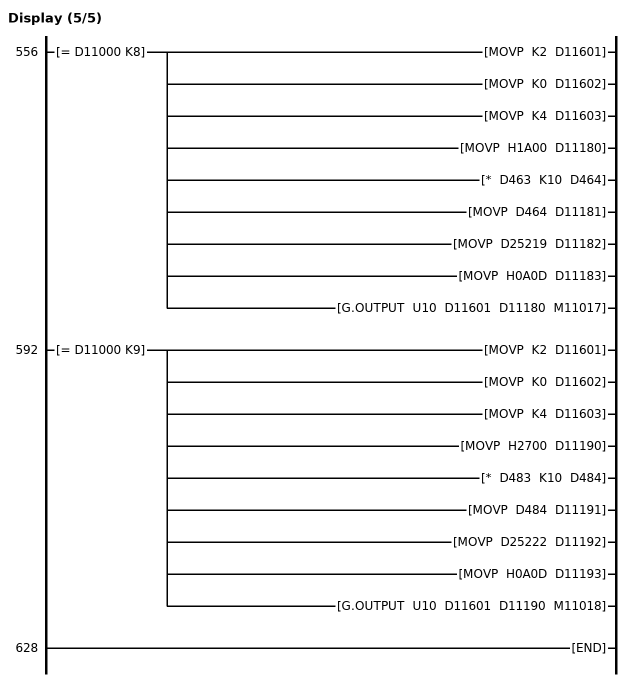
[picture p216: ladder of Display, rungs at steps 556 to 628]
556   LD=     D11000 K8
      MOVP    K2 D11601
      MOVP    K0 D11602
      MOVP    K4 D11603
      MOVP    H1A00 D11180
      *       D463 K10 D464
      MOVP    D464 D11181
      MOVP    D25219 D11182
      MOVP    H0A0D D11183
      G.OUTPUT U10 D11601 D11180 M11017
592   LD=     D11000 K9
      MOVP    K2 D11601
      MOVP    K0 D11602
      MOVP    K4 D11603
      MOVP    H2700 D11190
      *       D483 K10 D484
      MOVP    D484 D11191
      MOVP    D25222 D11192
      MOVP    H0A0D D11193
      G.OUTPUT U10 D11601 D11190 M11018
628   END
END_PROGRAM

PROGRAM door
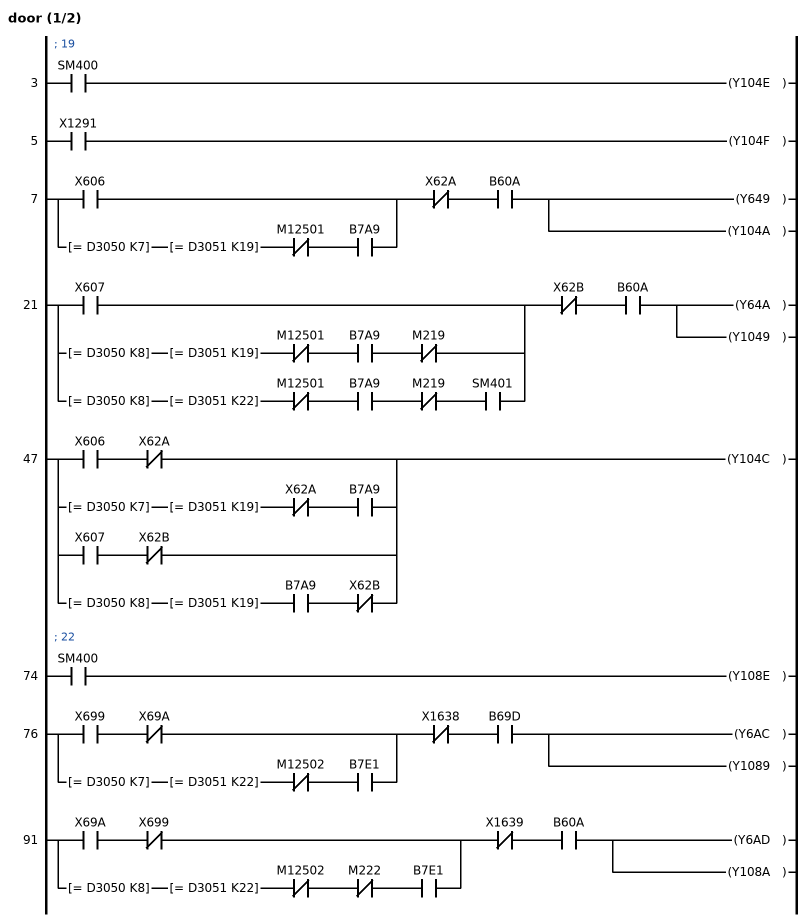
; 19
3     LD      SM400
      OUT     Y104E
5     LD      X1291
      OUT     Y104F
7     LD      X606
      LD=     D3050 K7
      AND=    D3051 K19
      ANI     M12501
      AND     B7A9
      ORB
      ANI     X62A
      AND     B60A
      OUT     Y649
      OUT     Y104A
21    LD      X607
      LD=     D3050 K8
      AND=    D3051 K19
      ANI     M12501
      AND     B7A9
      ANI     M219
      ORB
      LD=     D3050 K8
      AND=    D3051 K22
      ANI     M12501
      AND     B7A9
      ANI     M219
      AND     SM401
      ORB
      ANI     X62B
      AND     B60A
      OUT     Y64A
      OUT     Y1049
47    LD      X606
      ANI     X62A
      LD=     D3050 K7
      AND=    D3051 K19
      ANI     X62A
      AND     B7A9
      ORB
      LD      X607
      ANI     X62B
      ORB
      LD=     D3050 K8
      AND=    D3051 K19
      AND     B7A9
      ANI     X62B
      ORB
      OUT     Y104C
; 22
74    LD      SM400
      OUT     Y108E
76    LD      X699
      ANI     X69A
      LD=     D3050 K7
      AND=    D3051 K22
      ANI     M12502
      AND     B7E1
      ORB
      ANI     X1638
      AND     B69D
      OUT     Y6AC
      OUT     Y1089
91    LD      X69A
      ANI     X699
      LD=     D3050 K8
      AND=    D3051 K22
      ANI     M12502
      ANI     M222
      AND     B7E1
      ORB
      ANI     X1639
      AND     B60A
      OUT     Y6AD
      OUT     Y108A
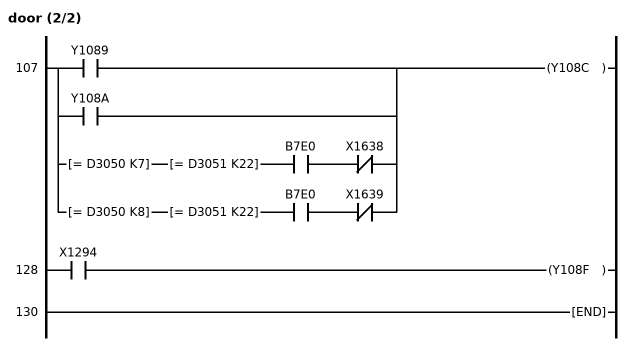
107   LD      Y1089
      OR      Y108A
      LD=     D3050 K7
      AND=    D3051 K22
      AND     B7E0
      ANI     X1638
      ORB
      LD=     D3050 K8
      AND=    D3051 K22
      AND     B7E0
      ANI     X1639
      ORB
      OUT     Y108C
128   LD      X1294
      OUT     Y108F
130   END
END_PROGRAM

PROGRAM enter_line
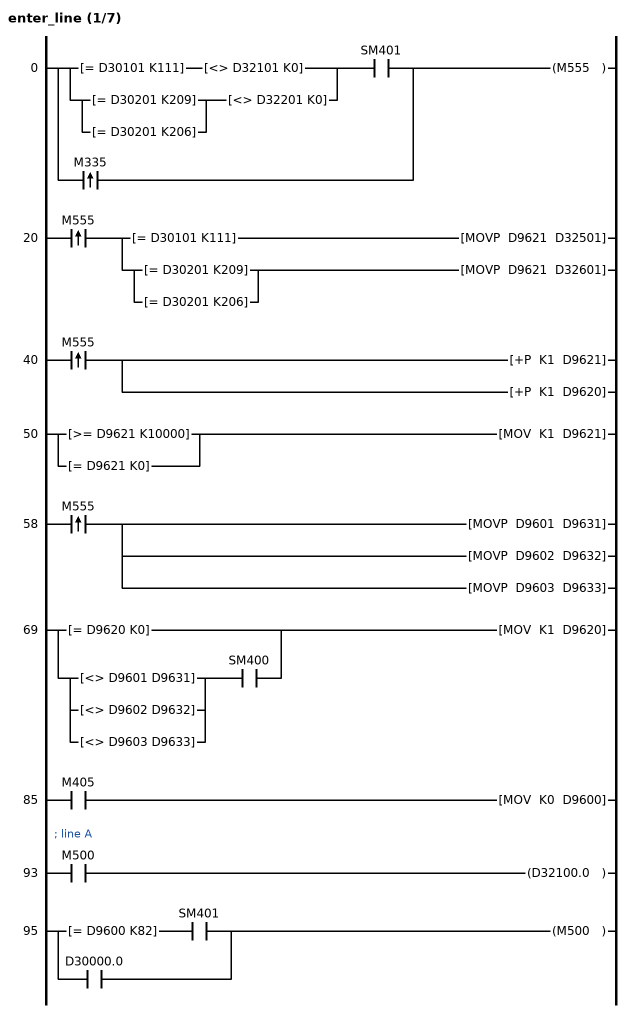
0     LD=     D30101 K111
      AND<>   D32101 K0
      LD=     D30201 K209
      OR=     D30201 K206
      AND<>   D32201 K0
      ORB
      AND     SM401
      ORP     M335
      OUT     M555
20    LDP     M555
      MPS
      AND=    D30101 K111
      MOVP    D9621 D32501
      MPP
      LD=     D30201 K209
      OR=     D30201 K206
      ANB
      MOVP    D9621 D32601
40    LDP     M555
      +P      K1 D9621
      +P      K1 D9620
50    LD>=    D9621 K10000
      OR=     D9621 K0
      MOV     K1 D9621
58    LDP     M555
      MOVP    D9601 D9631
      MOVP    D9602 D9632
      MOVP    D9603 D9633
69    LD=     D9620 K0
      LD<>    D9601 D9631
      OR<>    D9602 D9632
      OR<>    D9603 D9633
      AND     SM400
      ORB
      MOV     K1 D9620
85    LD      M405
      MOV     K0 D9600
; line A
93    LD      M500
      OUT     D32100.0
95    LD=     D9600 K82
      AND     SM401
      OR      D30000.0
      OUT     M500
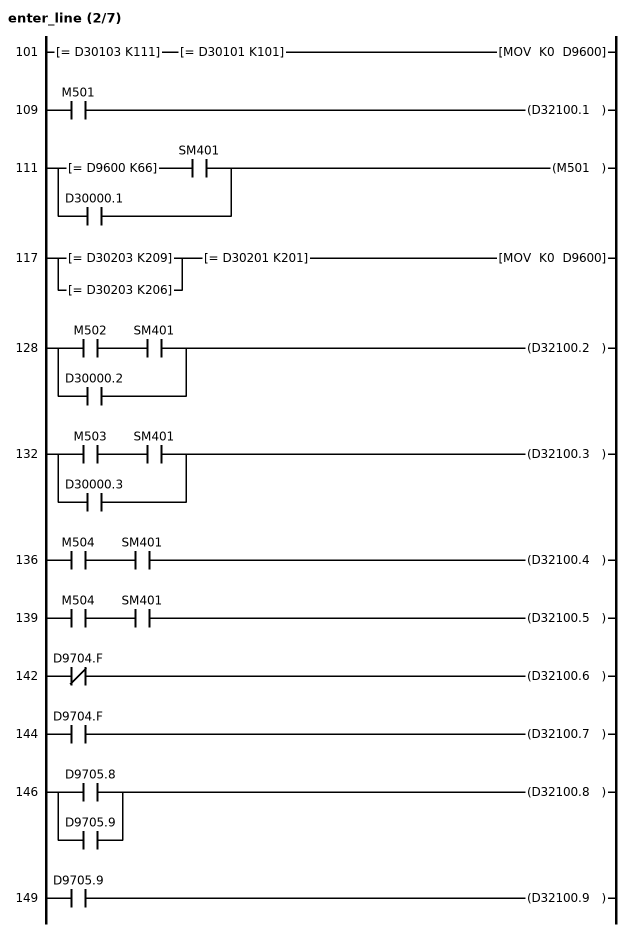
101   LD=     D30103 K111
      AND=    D30101 K101
      MOV     K0 D9600
109   LD      M501
      OUT     D32100.1
111   LD=     D9600 K66
      AND     SM401
      OR      D30000.1
      OUT     M501
117   LD=     D30203 K209
      OR=     D30203 K206
      AND=    D30201 K201
      MOV     K0 D9600
128   LD      M502
      AND     SM401
      OR      D30000.2
      OUT     D32100.2
132   LD      M503
      AND     SM401
      OR      D30000.3
      OUT     D32100.3
136   LD      M504
      AND     SM401
      OUT     D32100.4
139   LD      M504
      AND     SM401
      OUT     D32100.5
142   LDI     D9704.F
      OUT     D32100.6
144   LD      D9704.F
      OUT     D32100.7
146   LD      D9705.8
      OR      D9705.9
      OUT     D32100.8
149   LD      D9705.9
      OUT     D32100.9
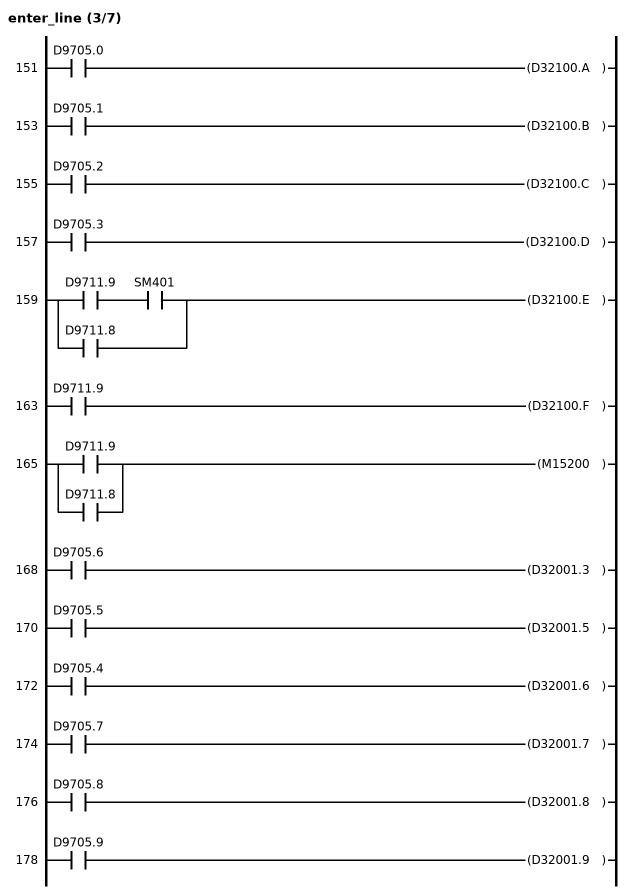
151   LD      D9705.0
      OUT     D32100.A
153   LD      D9705.1
      OUT     D32100.B
155   LD      D9705.2
      OUT     D32100.C
157   LD      D9705.3
      OUT     D32100.D
159   LD      D9711.9
      AND     SM401
      OR      D9711.8
      OUT     D32100.E
163   LD      D9711.9
      OUT     D32100.F
165   LD      D9711.9
      OR      D9711.8
      OUT     M15200
168   LD      D9705.6
      OUT     D32001.3
170   LD      D9705.5
      OUT     D32001.5
172   LD      D9705.4
      OUT     D32001.6
174   LD      D9705.7
      OUT     D32001.7
176   LD      D9705.8
      OUT     D32001.8
178   LD      D9705.9
      OUT     D32001.9
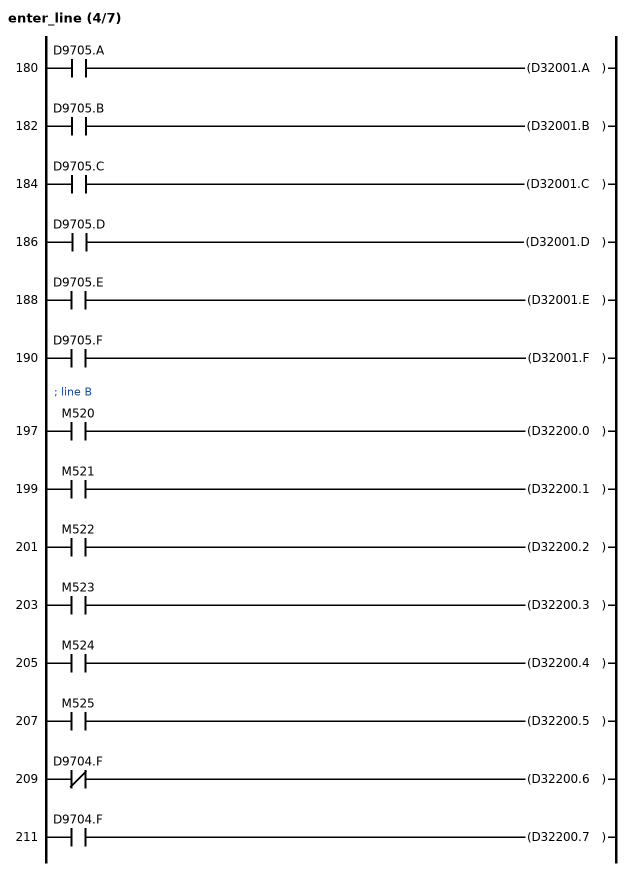
180   LD      D9705.A
      OUT     D32001.A
182   LD      D9705.B
      OUT     D32001.B
184   LD      D9705.C
      OUT     D32001.C
186   LD      D9705.D
      OUT     D32001.D
188   LD      D9705.E
      OUT     D32001.E
190   LD      D9705.F
      OUT     D32001.F
; line B
197   LD      M520
      OUT     D32200.0
199   LD      M521
      OUT     D32200.1
201   LD      M522
      OUT     D32200.2
203   LD      M523
      OUT     D32200.3
205   LD      M524
      OUT     D32200.4
207   LD      M525
      OUT     D32200.5
209   LDI     D9704.F
      OUT     D32200.6
211   LD      D9704.F
      OUT     D32200.7
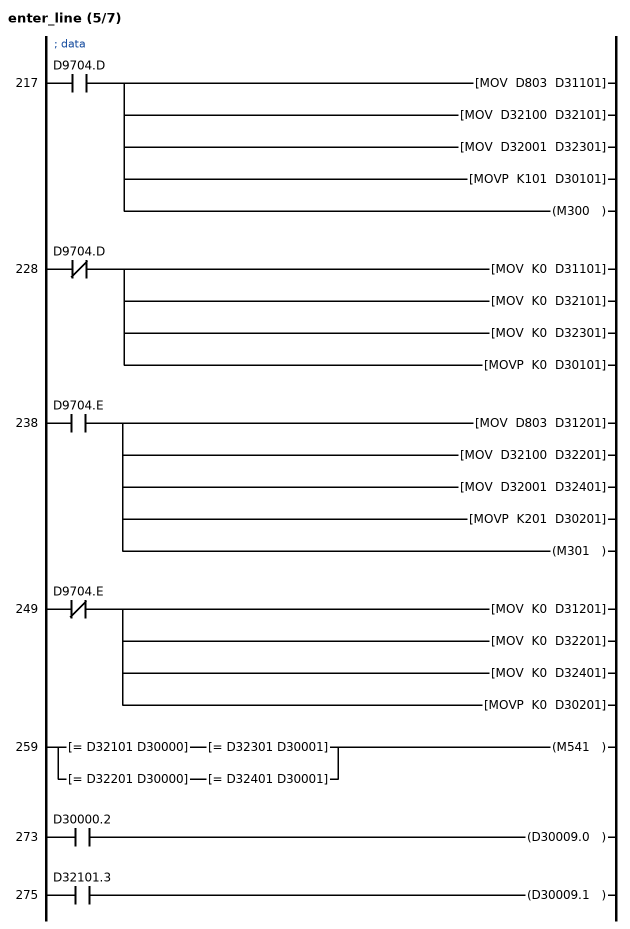
; data
217   LD      D9704.D
      MOV     D803 D31101
      MOV     D32100 D32101
      MOV     D32001 D32301
      MOVP    K101 D30101
      OUT     M300
228   LDI     D9704.D
      MOV     K0 D31101
      MOV     K0 D32101
      MOV     K0 D32301
      MOVP    K0 D30101
238   LD      D9704.E
      MOV     D803 D31201
      MOV     D32100 D32201
      MOV     D32001 D32401
      MOVP    K201 D30201
      OUT     M301
249   LDI     D9704.E
      MOV     K0 D31201
      MOV     K0 D32201
      MOV     K0 D32401
      MOVP    K0 D30201
259   LD=     D32101 D30000
      AND=    D32301 D30001
      LD=     D32201 D30000
      AND=    D32401 D30001
      ORB
      OUT     M541
273   LD      D30000.2
      OUT     D30009.0
275   LD      D32101.3
      OUT     D30009.1
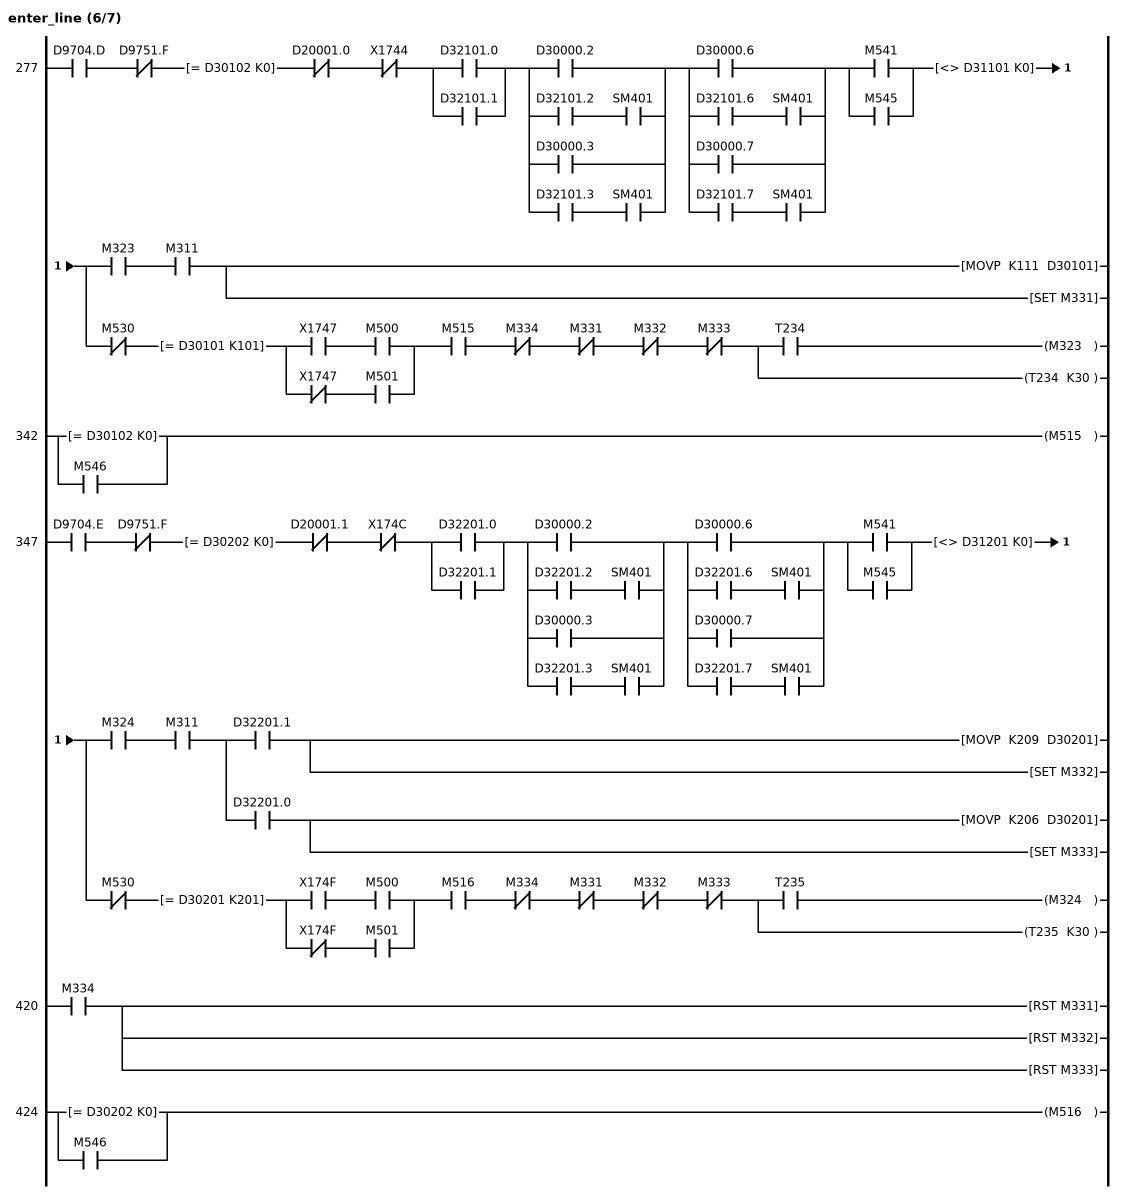
277   LD      D9704.D
      ANI     D9751.F
      AND=    D30102 K0
      ANI     D20001.0
      ANI     X1744
      LD      D32101.0
      OR      D32101.1
      ANB
      LD      D30000.2
      LD      D32101.2
      AND     SM401
      ORB
      OR      D30000.3
      LD      D32101.3
      AND     SM401
      ORB
      ANB
      LD      D30000.6
      LD      D32101.6
      AND     SM401
      ORB
      OR      D30000.7
      LD      D32101.7
      AND     SM401
      ORB
      ANB
      LD      M541
      OR      M545
      ANB
      AND<>   D31101 K0
      MPS
      AND     M323
      AND     M311
      MOVP    K111 D30101
      SET     M331
      MPP
      ANI     M530
      AND=    D30101 K101
      LD      X1747
      AND     M500
      LDI     X1747
      AND     M501
      ORB
      ANB
      AND     M515
      ANI     M334
      ANI     M331
      ANI     M332
      ANI     M333
      MPS
      AND     T234
      OUT     M323
      MPP
      OUT     T234 K30
342   LD=     D30102 K0
      OR      M546
      OUT     M515
347   LD      D9704.E
      ANI     D9751.F
      AND=    D30202 K0
      ANI     D20001.1
      ANI     X174C
      LD      D32201.0
      OR      D32201.1
      ANB
      LD      D30000.2
      LD      D32201.2
      AND     SM401
      ORB
      OR      D30000.3
      LD      D32201.3
      AND     SM401
      ORB
      ANB
      LD      D30000.6
      LD      D32201.6
      AND     SM401
      ORB
      OR      D30000.7
      LD      D32201.7
      AND     SM401
      ORB
      ANB
      LD      M541
      OR      M545
      ANB
      AND<>   D31201 K0
      MPS
      AND     M324
      AND     M311
      MPS
      AND     D32201.1
      MOVP    K209 D30201
      SET     M332
      MPP
      AND     D32201.0
      MOVP    K206 D30201
      SET     M333
      MPP
      ANI     M530
      AND=    D30201 K201
      LD      X174F
      AND     M500
      LDI     X174F
      AND     M501
      ORB
      ANB
      AND     M516
      ANI     M334
      ANI     M331
      ANI     M332
      ANI     M333
      MPS
      AND     T235
      OUT     M324
      MPP
      OUT     T235 K30
420   LD      M334
      RST     M331
      RST     M332
      RST     M333
424   LD=     D30202 K0
      OR      M546
      OUT     M516
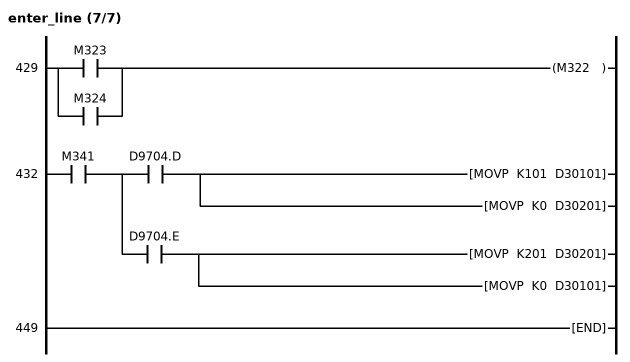
429   LD      M323
      OR      M324
      OUT     M322
432   LD      M341
      MPS
      AND     D9704.D
      MOVP    K101 D30101
      MOVP    K0 D30201
      MPP
      AND     D9704.E
      MOVP    K201 D30201
      MOVP    K0 D30101
449   END
END_PROGRAM

FUNCTION_BLOCK I+ST_9118b3cfc5d74fe4
VAR_INPUT
  __IST_EN_IN : BOOL;
END_VAR
VAR_OUTPUT
  __IST_EN_OUT : BOOL;
END_VAR
(* IST HEADER START *)
IF NOT __IST_EN_IN THEN __IST_EN_OUT:=FALSE; RETURN; END_IF;
(* VERSION=1:TYPE=STB *)
(* IST HEADER END *)
D7313:=D7311+D7312+D7314;
D913:=D7313;

D7317:=D7315+D7316+D7318;
D917:=D7317;

D7321:=D7319+D7320+D7322;
D921:=D7321;

D7325:=D7323+D7324+D7326;
D925:=D7325;
END_FUNCTION_BLOCK

PROGRAM input
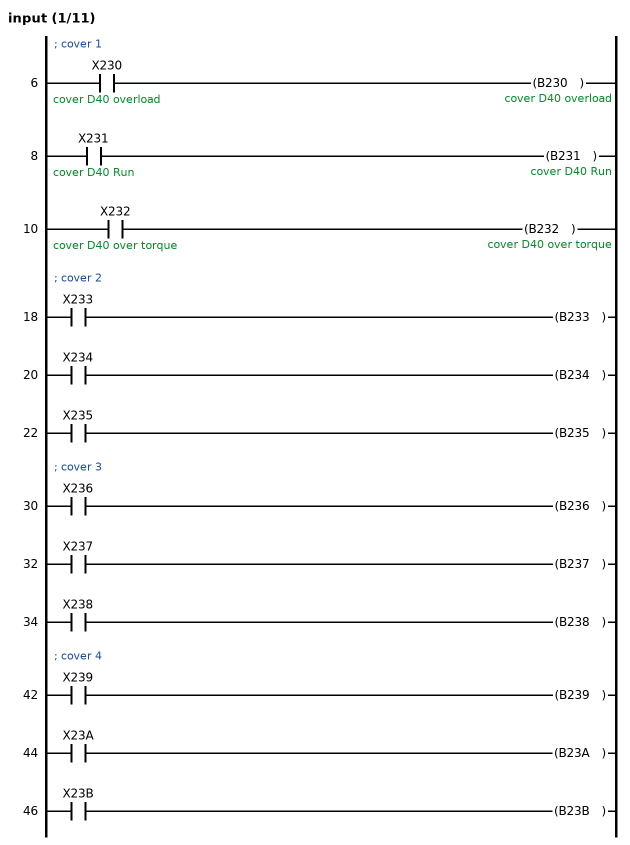
; cover 1
6     LD      X230  ; cover D40 overload
      OUT     B230  ; cover D40 overload
8     LD      X231  ; cover D40 Run
      OUT     B231  ; cover D40 Run
10    LD      X232  ; cover D40 over torque
      OUT     B232  ; cover D40 over torque
; cover 2
18    LD      X233
      OUT     B233
20    LD      X234
      OUT     B234
22    LD      X235
      OUT     B235
; cover 3
30    LD      X236
      OUT     B236
32    LD      X237
      OUT     B237
34    LD      X238
      OUT     B238
; cover 4
42    LD      X239
      OUT     B239
44    LD      X23A
      OUT     B23A
46    LD      X23B
      OUT     B23B
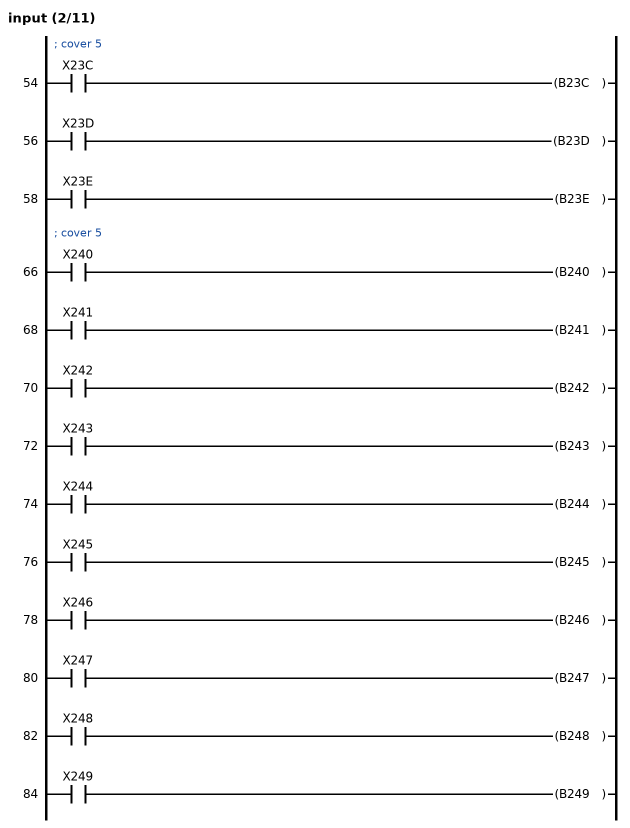
; cover 5
54    LD      X23C
      OUT     B23C
56    LD      X23D
      OUT     B23D
58    LD      X23E
      OUT     B23E
; cover 5
66    LD      X240
      OUT     B240
68    LD      X241
      OUT     B241
70    LD      X242
      OUT     B242
72    LD      X243
      OUT     B243
74    LD      X244
      OUT     B244
76    LD      X245
      OUT     B245
78    LD      X246
      OUT     B246
80    LD      X247
      OUT     B247
82    LD      X248
      OUT     B248
84    LD      X249
      OUT     B249
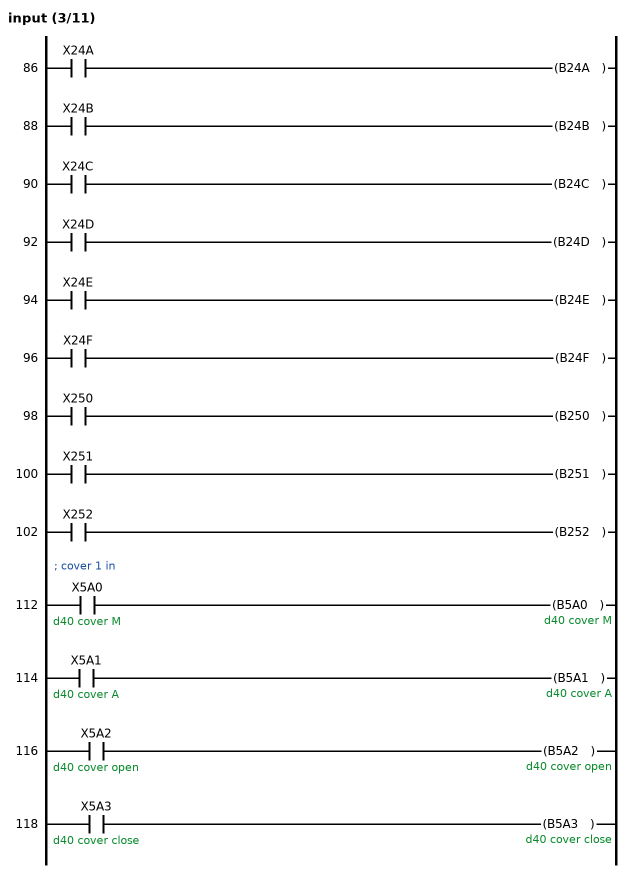
86    LD      X24A
      OUT     B24A
88    LD      X24B
      OUT     B24B
90    LD      X24C
      OUT     B24C
92    LD      X24D
      OUT     B24D
94    LD      X24E
      OUT     B24E
96    LD      X24F
      OUT     B24F
98    LD      X250
      OUT     B250
100   LD      X251
      OUT     B251
102   LD      X252
      OUT     B252
; cover 1 in
112   LD      X5A0  ; d40 cover M
      OUT     B5A0  ; d40 cover M
114   LD      X5A1  ; d40 cover A
      OUT     B5A1  ; d40 cover A
116   LD      X5A2  ; d40 cover open
      OUT     B5A2  ; d40 cover open
118   LD      X5A3  ; d40 cover close
      OUT     B5A3  ; d40 cover close
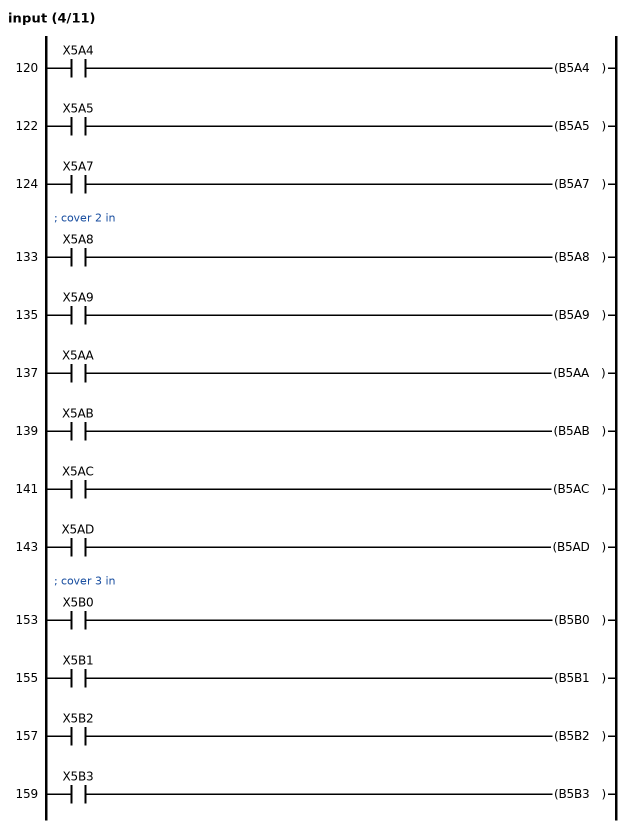
120   LD      X5A4
      OUT     B5A4
122   LD      X5A5
      OUT     B5A5
124   LD      X5A7
      OUT     B5A7
; cover 2 in
133   LD      X5A8
      OUT     B5A8
135   LD      X5A9
      OUT     B5A9
137   LD      X5AA
      OUT     B5AA
139   LD      X5AB
      OUT     B5AB
141   LD      X5AC
      OUT     B5AC
143   LD      X5AD
      OUT     B5AD
; cover 3 in
153   LD      X5B0
      OUT     B5B0
155   LD      X5B1
      OUT     B5B1
157   LD      X5B2
      OUT     B5B2
159   LD      X5B3
      OUT     B5B3
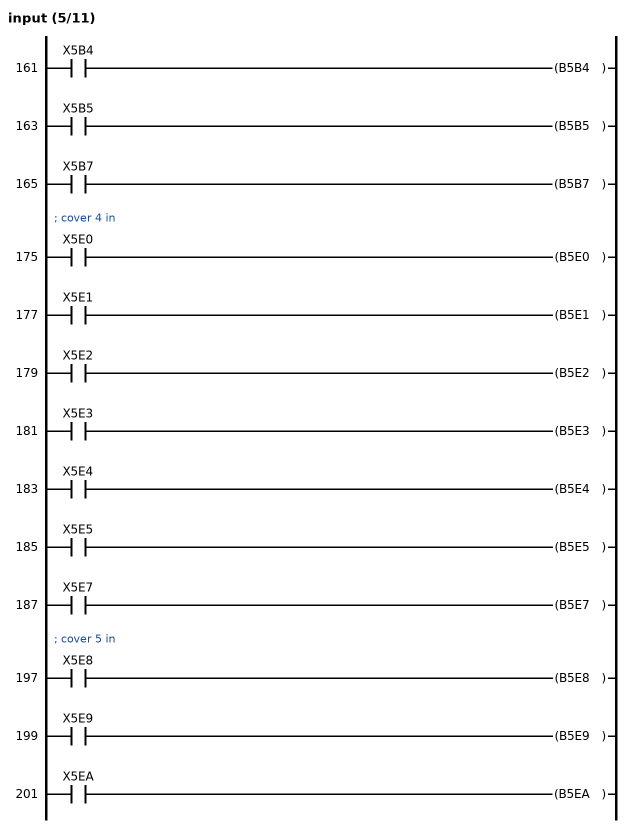
161   LD      X5B4
      OUT     B5B4
163   LD      X5B5
      OUT     B5B5
165   LD      X5B7
      OUT     B5B7
; cover 4 in
175   LD      X5E0
      OUT     B5E0
177   LD      X5E1
      OUT     B5E1
179   LD      X5E2
      OUT     B5E2
181   LD      X5E3
      OUT     B5E3
183   LD      X5E4
      OUT     B5E4
185   LD      X5E5
      OUT     B5E5
187   LD      X5E7
      OUT     B5E7
; cover 5 in
197   LD      X5E8
      OUT     B5E8
199   LD      X5E9
      OUT     B5E9
201   LD      X5EA
      OUT     B5EA
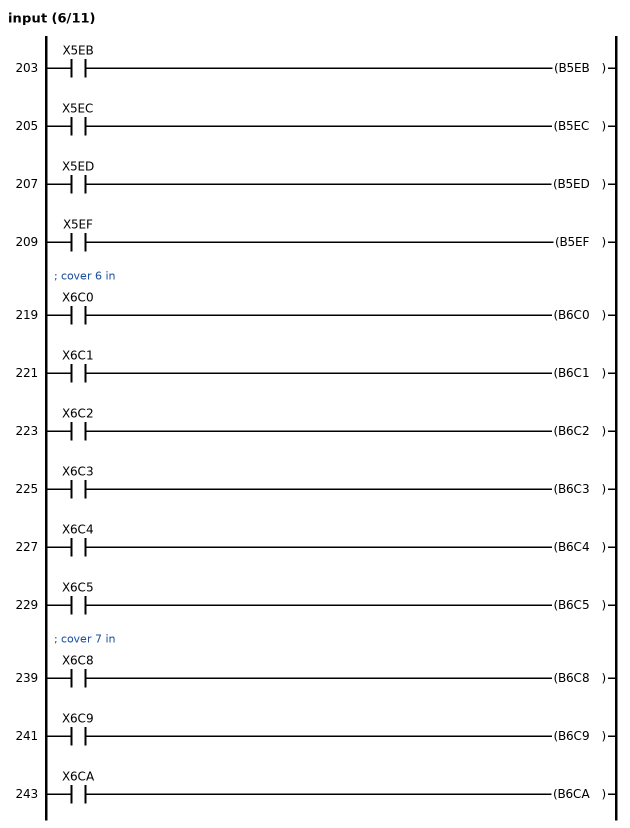
203   LD      X5EB
      OUT     B5EB
205   LD      X5EC
      OUT     B5EC
207   LD      X5ED
      OUT     B5ED
209   LD      X5EF
      OUT     B5EF
; cover 6 in
219   LD      X6C0
      OUT     B6C0
221   LD      X6C1
      OUT     B6C1
223   LD      X6C2
      OUT     B6C2
225   LD      X6C3
      OUT     B6C3
227   LD      X6C4
      OUT     B6C4
229   LD      X6C5
      OUT     B6C5
; cover 7 in
239   LD      X6C8
      OUT     B6C8
241   LD      X6C9
      OUT     B6C9
243   LD      X6CA
      OUT     B6CA
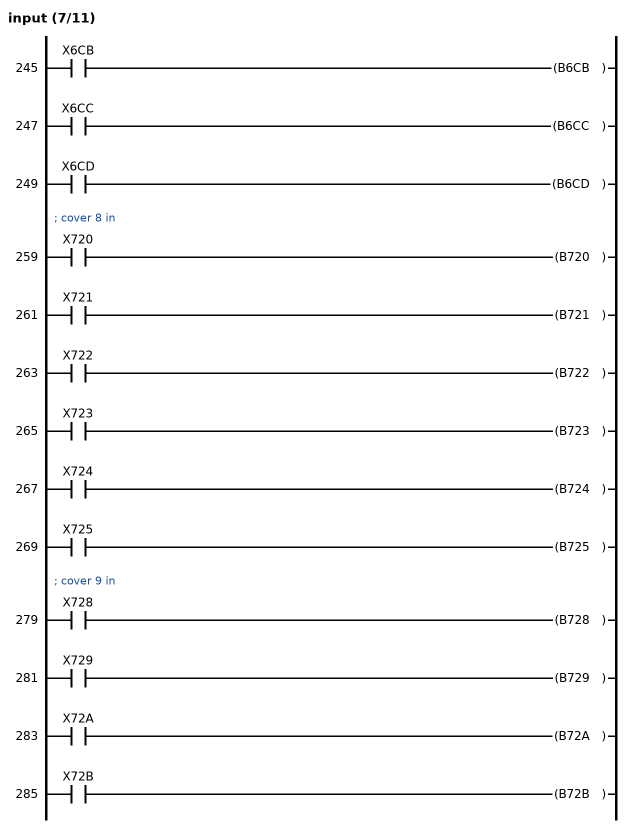
245   LD      X6CB
      OUT     B6CB
247   LD      X6CC
      OUT     B6CC
249   LD      X6CD
      OUT     B6CD
; cover 8 in
259   LD      X720
      OUT     B720
261   LD      X721
      OUT     B721
263   LD      X722
      OUT     B722
265   LD      X723
      OUT     B723
267   LD      X724
      OUT     B724
269   LD      X725
      OUT     B725
; cover 9 in
279   LD      X728
      OUT     B728
281   LD      X729
      OUT     B729
283   LD      X72A
      OUT     B72A
285   LD      X72B
      OUT     B72B
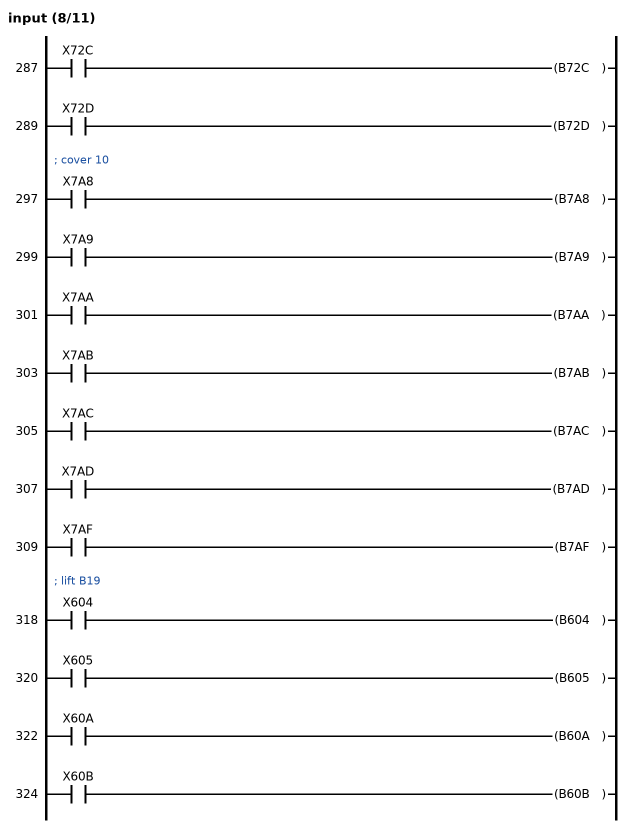
287   LD      X72C
      OUT     B72C
289   LD      X72D
      OUT     B72D
; cover 10
297   LD      X7A8
      OUT     B7A8
299   LD      X7A9
      OUT     B7A9
301   LD      X7AA
      OUT     B7AA
303   LD      X7AB
      OUT     B7AB
305   LD      X7AC
      OUT     B7AC
307   LD      X7AD
      OUT     B7AD
309   LD      X7AF
      OUT     B7AF
; lift B19
318   LD      X604
      OUT     B604
320   LD      X605
      OUT     B605
322   LD      X60A
      OUT     B60A
324   LD      X60B
      OUT     B60B
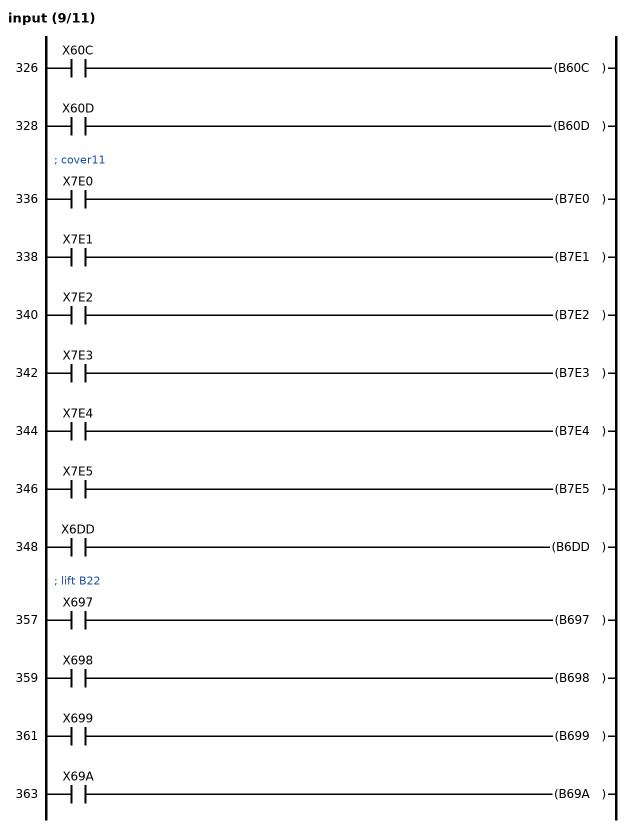
326   LD      X60C
      OUT     B60C
328   LD      X60D
      OUT     B60D
; cover11
336   LD      X7E0
      OUT     B7E0
338   LD      X7E1
      OUT     B7E1
340   LD      X7E2
      OUT     B7E2
342   LD      X7E3
      OUT     B7E3
344   LD      X7E4
      OUT     B7E4
346   LD      X7E5
      OUT     B7E5
348   LD      X6DD
      OUT     B6DD
; lift B22
357   LD      X697
      OUT     B697
359   LD      X698
      OUT     B698
361   LD      X699
      OUT     B699
363   LD      X69A
      OUT     B69A
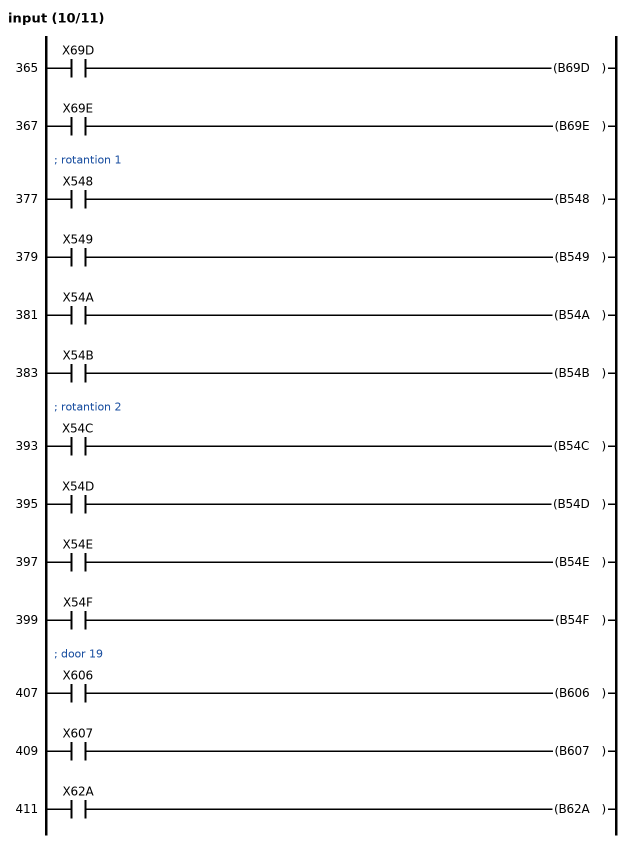
365   LD      X69D
      OUT     B69D
367   LD      X69E
      OUT     B69E
; rotantion 1
377   LD      X548
      OUT     B548
379   LD      X549
      OUT     B549
381   LD      X54A
      OUT     B54A
383   LD      X54B
      OUT     B54B
; rotantion 2
393   LD      X54C
      OUT     B54C
395   LD      X54D
      OUT     B54D
397   LD      X54E
      OUT     B54E
399   LD      X54F
      OUT     B54F
; door 19
407   LD      X606
      OUT     B606
409   LD      X607
      OUT     B607
411   LD      X62A
      OUT     B62A
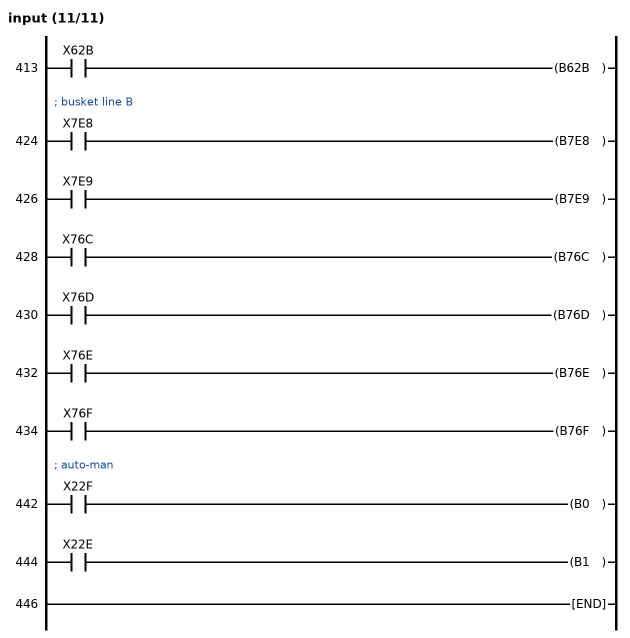
413   LD      X62B
      OUT     B62B
; busket line B
424   LD      X7E8
      OUT     B7E8
426   LD      X7E9
      OUT     B7E9
428   LD      X76C
      OUT     B76C
430   LD      X76D
      OUT     B76D
432   LD      X76E
      OUT     B76E
434   LD      X76F
      OUT     B76F
; auto-man
442   LD      X22F
      OUT     B0
444   LD      X22E
      OUT     B1
446   END
END_PROGRAM

PROGRAM lift
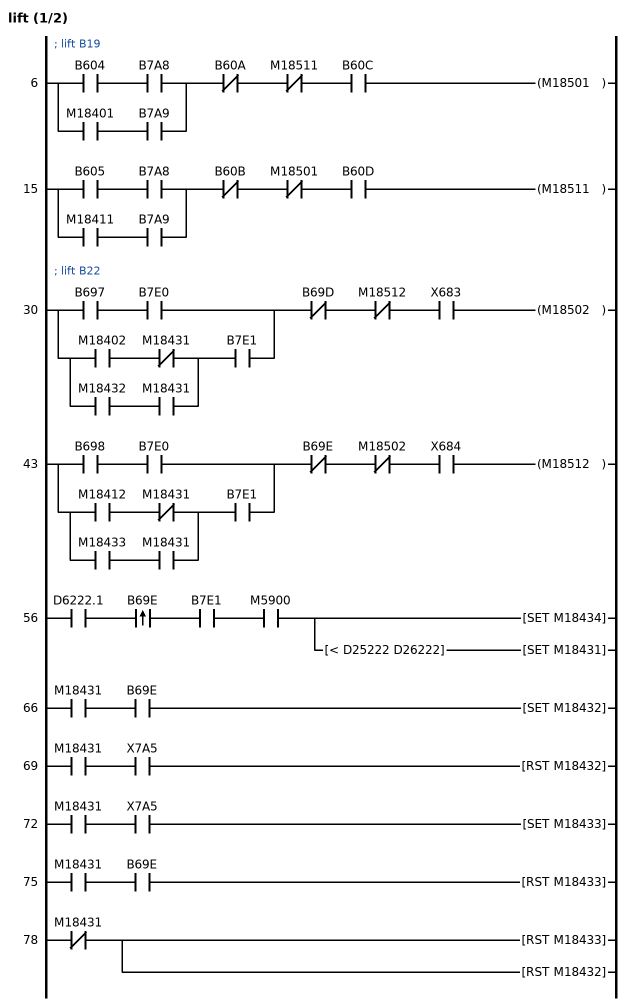
; lift B19
6     LD      B604
      AND     B7A8
      LD      M18401
      AND     B7A9
      ORB
      ANI     B60A
      ANI     M18511
      AND     B60C
      OUT     M18501
15    LD      B605
      AND     B7A8
      LD      M18411
      AND     B7A9
      ORB
      ANI     B60B
      ANI     M18501
      AND     B60D
      OUT     M18511
; lift B22
30    LD      B697
      AND     B7E0
      LD      M18402
      ANI     M18431
      LD      M18432
      AND     M18431
      ORB
      AND     B7E1
      ORB
      ANI     B69D
      ANI     M18512
      AND     X683
      OUT     M18502
43    LD      B698
      AND     B7E0
      LD      M18412
      ANI     M18431
      LD      M18433
      AND     M18431
      ORB
      AND     B7E1
      ORB
      ANI     B69E
      ANI     M18502
      AND     X684
      OUT     M18512
56    LD      D6222.1
      ANDP    B69E
      AND     B7E1
      AND     M5900
      SET     M18434
      AND<    D25222 D26222
      SET     M18431
66    LD      M18431
      AND     B69E
      SET     M18432
69    LD      M18431
      AND     X7A5
      RST     M18432
72    LD      M18431
      AND     X7A5
      SET     M18433
75    LD      M18431
      AND     B69E
      RST     M18433
78    LDI     M18431
      RST     M18433
      RST     M18432
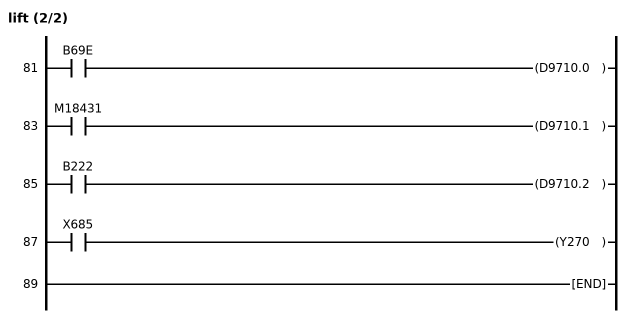
81    LD      B69E
      OUT     D9710.0
83    LD      M18431
      OUT     D9710.1
85    LD      B222
      OUT     D9710.2
87    LD      X685
      OUT     Y270
89    END
END_PROGRAM

PROGRAM lift_door_step
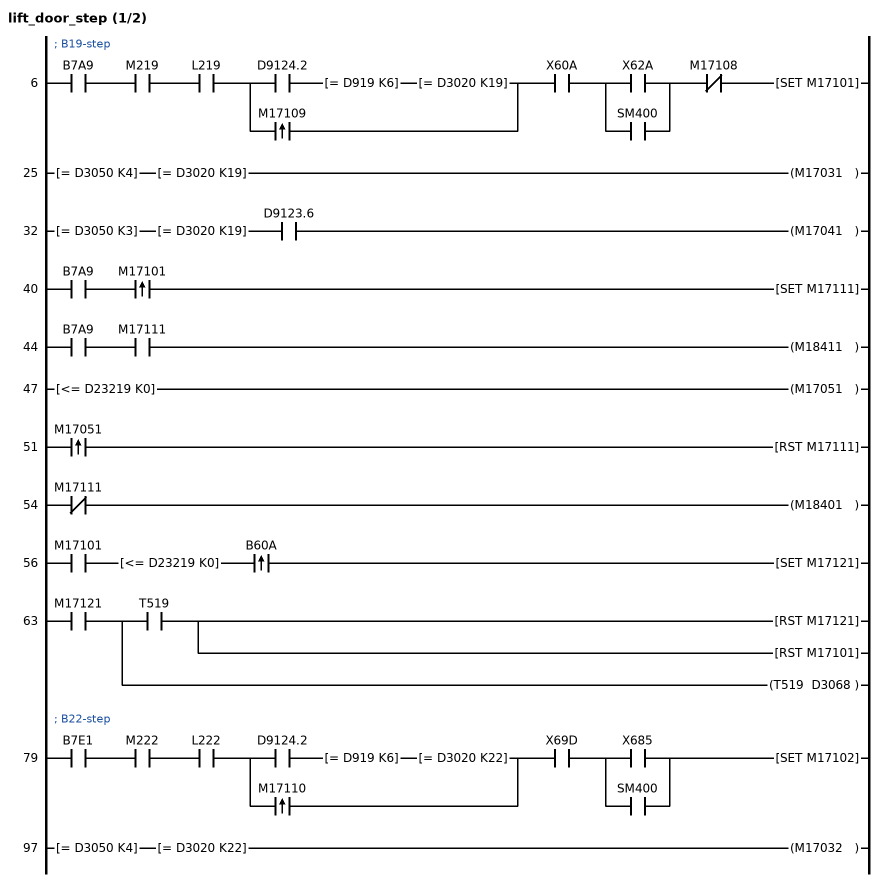
; B19-step
6     LD      B7A9
      AND     M219
      AND     L219
      LD      D9124.2
      AND=    D919 K6
      AND=    D3020 K19
      ORP     M17109
      ANB
      AND     X60A
      LD      X62A
      OR      SM400
      ANB
      ANI     M17108
      SET     M17101
25    LD=     D3050 K4
      AND=    D3020 K19
      OUT     M17031
32    LD=     D3050 K3
      AND=    D3020 K19
      AND     D9123.6
      OUT     M17041
40    LD      B7A9
      ANDP    M17101
      SET     M17111
44    LD      B7A9
      AND     M17111
      OUT     M18411
47    LD<=    D23219 K0
      OUT     M17051
51    LDP     M17051
      RST     M17111
54    LDI     M17111
      OUT     M18401
56    LD      M17101
      AND<=   D23219 K0
      ANDP    B60A
      SET     M17121
63    LD      M17121
      MPS
      AND     T519
      RST     M17121
      RST     M17101
      MPP
      OUT     T519 D3068
; B22-step
79    LD      B7E1
      AND     M222
      AND     L222
      LD      D9124.2
      AND=    D919 K6
      AND=    D3020 K22
      ORP     M17110
      ANB
      AND     X69D
      LD      X685
      OR      SM400
      ANB
      SET     M17102
97    LD=     D3050 K4
      AND=    D3020 K22
      OUT     M17032
